// TwinCAT 3 PLC project PLC
// ProgramVersion: 3.1.4024.0
// libraries:
//   Tc2_Standard, * (Beckhoff Automation GmbH)
//   Tc2_System, * (Beckhoff Automation GmbH)
//   Tc3_Module, * (Beckhoff Automation GmbH)
// project tree:
//   / PlcTask.TcTTO
//   POUs/ FB_Count.TcPOU, MAIN.TcPOU
// real-time tasks:
//   TASK PlcTask: cycle T#10ms, priority 20, ADS port 350
//   TASK PlcTask1: cycle T#10ms, priority 21, ADS port 351
// I/O:
//   DEVICE Device 1 (EtherCAT), AmsNetId 0.0.0.0.2.1
//     Term 1 (EK1200) [EK1200-5000 EtherCAT Power supply (2A E-Bus)]
//       Term 2 (EL1859) [EL1859 8Ch. Dig. Input 24V, 3ms, 8Ch. Dig. Output 24V, 0.5A]
//       Term 3 (EL3702) [EL3702 2Ch. Ana. Input +/-10V, DIFF, Oversample]
//       Term 4 (EL4032) [EL4032 2Ch. Ana. Output +/-10V, 12bit]
//       Term 5 (EL3201) [EL3201 1Ch. Ana. Input PT100 (RTD)]
//       Term 6 (EL9011) [EL9011 End Terminal]
// variable links:
//   PLC Instance <-> Device 1 (EtherCAT)/Term 1 (EK1200)/Term 2 (EL1859)
//     PlcTask Outputs/MAIN.bLed{1..4} <-> Channel {9..12}/Output  (4 links)

CONFIGURATION PLC
    RESOURCE PLC ON TwinCAT3
        TASK PlcTask(INTERVAL := T#10ms, PRIORITY := 20);
        PROGRAM MAIN WITH PlcTask : MAIN;
    END_RESOURCE
END_CONFIGURATION

// ---- POUs/MAIN.TcPOU
PROGRAM MAIN
VAR
	fbCount		: FB_Count;
	bCount		: BOOL;
	nCounter	: INT;
	nCounter2	: INT;
	nCounter3	: INT;
	
	bLed1	AT %Q*	: BOOL;
	bLed2	AT %Q*	: BOOL;
	bLed3	AT %Q*	: BOOL;
	bLed4	AT %Q*	: BOOL;
	
END_VAR

fbCount(
	bCount			:= bCount,
	nCountIncrement	:= 2
//	nCounterValue	=> nCounter
);

nCounter := nCounter +1;

IF nCounter MOD 20 = 0 THEN

{IF defined (Variant1)}
	bLed3 := nCounter.2;
	bLed4 := nCounter.3;
{ELSE}
	bLed1 := nCounter.2;
	bLed2 := nCounter.3;
{END_IF}



END_IF

END_PROGRAM

// ---- POUs/FB_Count.TcPOU
FUNCTION_BLOCK FB_Count
VAR_INPUT
	bCount 			: BOOL;
	nCountIncrement : INT := 1;
END_VAR
VAR_OUTPUT
	nCounterValue : INT;
END_VAR
VAR
	rtCount : R_TRIG;
END_VAR

rtCount(CLK := bCount);
IF rtCount.Q THEN
	nCounterValue := nCounterValue + nCountIncrement;
END_IF

END_FUNCTION_BLOCK
